PROGRAM TorqueCounnter
VAR
	startTest: BOOL:=FALSE;
	i :INT:=1;
	Torque_Nm: INT:=5;
	j: INT:=14;
	TorqueCounter: INT:=0;
	TorqInterval  : INT:=100;
	n: INT;
END_VAR

IF startTest THEN
				TorqueCounter := TorqueCounter + 1;
				
				IF   TorqueCounter >= TorqInterval*(i-1) AND TorqueCounter <TorqInterval*i THEN
					 IF i<=j/2 THEN
						FOR i:=1 TO j/2 BY 1 DO	
							
								IF i MOD 2=1 THEN
								link.torqueX := TO_INT(Torque_Nm * i/2.37*1000);
								ELSE
								link.torqueX := TO_INT(-Torque_Nm * i/2.37*1000);	
	 							END_IF
								
							
						 END_FOR
					   ELSIF i>j/2 THEN
	  					FOR i:=j TO j/2 BY -1 DO	
							IF i MOD 2=1 THEN
								link.torqueX := TO_INT(Torque_Nm * i/2.37*1000);
							ELSE
								link.torqueX := TO_INT(-Torque_Nm * i/2.37*1000);	
	 						END_IF							
						 END_FOR
						
					END_IF					
					
				END_IF				
						
			ELSE
		link.torqueX := 0;
		startTest := FALSE;
		TorqueCounter := 0; 	
END_IF

END_PROGRAM

(* stored: Version 1.1.0.1, ProductVersion 3.1.4024.9
   POU TorqueCounnter: Id {11272ec1-26bf-41ff-be6d-e0596e66524e}, SpecialFunc None *)
